// TIA Portal V17 export
// export: Created 2025-08-05T09:36:00.6518849Z, ExportSetting WithDefaults, DisplayName Totally Integrated Automation Portal, DisplayVersion V17, DisplayName TIA Portal Openness, DisplayVersion V17, DisplayName TIA Portal Version Control Interface, DisplayVersion V17, DisplayName SINAMICS Startdrive Advanced, DisplayVersion V17, DisplayName SINAMICS Startdrive G130, G150, S120, S150, SINAMICS MV, S210, DisplayVersion V17, DisplayName SINAMICS Startdrive G110M, G120, G120C, G120D, G120P, G115D, DisplayVersion V17, DisplayName STEP 7 Professional, DisplayVersion V17, DisplayName STEP 7 Safety, DisplayVersion V17, DisplayName WinCC Advanced, DisplayVersion V17
TYPE "typeMSOs"
// stored: IsFailsafeCompliant false
   STRUCT
      activeMSO2 : Bool;   // Betriebsart 2 aktiv + Zustimmtaster gedrückt
      activeMSO3 : Bool;   // Betriebsart 3 aktiv + Zustimmtaster gedrückt
      selectedMSO2 : Bool;   // Betriebsart 2 angewählt
      selectedMSO3 : Bool;   // Betriebsart 3 angewählt
   END_STRUCT;
END_TYPE
